# EPICS autosave request: iocBoot/ioc13MARCCD2/auto_settings.req
file "marCCD_settings.req",       P=$(P),  R=cam1:
file "NDStdArrays_settings.req",  P=$(P),  R=image1:
file "commonPlugin_settings.req", P=$(P)
